FUNCTION_BLOCK Crane EXTENDS BaseCarrier
VAR_INPUT
END_VAR
VAR_OUTPUT
	o_VacuumGripper: VacuumGripper;
	o_MonostableCylinder: MonostableCylinder;
END_VAR
VAR
	// Turning table
	m_PresenceSensorAtStack : PresenceSensor;
	m_PresenceSensorAtConveyor : PresenceSensor;
	m_PresenceSensorAtStamp : PresenceSensor;
END_VAR

PROPERTY AtConveyor : BOOL
GET
AtConveyor := m_PresenceSensorAtConveyor.Value;
END_GET
END_PROPERTY

PROPERTY AtStack : BOOL
GET
AtStack := m_PresenceSensorAtStack.Value;
END_GET
END_PROPERTY

PROPERTY AtStamp : BOOL
GET
AtStamp := m_PresenceSensorAtStamp.Value;
END_GET
END_PROPERTY

METHOD METH_CarrierStop : BOOL
VAR_INPUT
END_VAR
Motor.ACT_Stop();
END_METHOD

METHOD METH_CarrierTurnClockwise : BOOL
VAR_INPUT
END_VAR
Motor.ACT_TurnClockwise();
END_METHOD

METHOD METH_CarrierTurnCounterclockwise : BOOL
VAR_INPUT
END_VAR
Motor.ACT_TurnCounterclockwise();
END_METHOD

END_FUNCTION_BLOCK

(* stored: Version 1.1.0.1
   POU Crane: Id {d5a70bf2-bda5-4136-8603-338529bb4c08}, SpecialFunc None
   Property AtConveyor: Id {2f4a99f8-e33c-40a7-92fe-e16a9bc15ea4}
   Get Get: Id {dc3d1ab7-bf1a-41c8-949c-6ac6c48d0d21}
   Property AtStack: Id {5ac6d5fd-9f88-46e3-9591-8e5ecde6851c}
   Get Get: Id {21f14694-4b73-4895-9cfc-a6ef7633e376}
   Property AtStamp: Id {a08342aa-263a-4577-93dc-0e209b4e221b}
   Get Get: Id {79e4e319-1e57-40d0-ab59-ada5d5c07cac}
   Method METH_CarrierStop: Id {598df988-4e64-4984-94c3-aedb5010aa2d}
   Method METH_CarrierTurnClockwise: Id {39fb0bf5-69df-4601-a397-176393e88b5b}
   Method METH_CarrierTurnCounterclockwise: Id {68209966-43a8-409a-a01d-a2236b832132} *)
